// TIA Portal V19 program export: 1 tag tables, 1 data types, 3 data blocks, 8 code blocks (in call order from the OBs), 17 instance data blocks

VAR_GLOBAL   // PLC tag table "Default tag table"
   B0 AT %QB0 : Byte;
   B1 AT %QB1 : Byte;
   Clock_Byte AT %MB0 : Byte;
   Clock_10Hz AT %M0.0 : Bool;
   Clock_5Hz AT %M0.1 : Bool;
   "Clock_2.5Hz" AT %M0.2 : Bool;
   Clock_2Hz AT %M0.3 : Bool;
   "Clock_1.25Hz" AT %M0.4 : Bool;
   Clock_1Hz AT %M0.5 : Bool;
   "Clock_0.625Hz" AT %M0.6 : Bool;
   "Clock_0.5Hz" AT %M0.7 : Bool;
   System_Byte AT %MB1 : Byte;
   FirstScan AT %M1.0 : Bool;
   DiagStatusUpdate AT %M1.1 : Bool;
   AlwaysTRUE AT %M1.2 : Bool;
   AlwaysFALSE AT %M1.3 : Bool;
   "from et200sp PLC_1" AT %IB100 : Byte;
   toET200spfromPLC1 AT %QB100 : Byte;
   "from et200sp PLC_1 Right" AT %IB200 : Byte;
   "toET200spfromPLC1 Right" AT %QB200 : Byte;
END_VAR

TYPE "NetworkSwitchHMI"
   STRUCT
      Ports { S7_SetPoint := 'True'} : Array[1..8] of "LPNDR_typePortInformation";
      Port { S7_SetPoint := 'True'} : "LPNDR_typePortInformation";
      Index { S7_SetPoint := 'True'} : Int := 1;
   END_STRUCT;
END_TYPE

DATA_BLOCK "GlobalDB"   // DB9
{ S7_Optimized_Access := 'FALSE' }
   VAR RETAIN
      RTInfo : Struct   // Used to collect runtime information on an individual FB/FC
         Mode : UInt := 1;
         OBnumber : OB_ANY := 1;
         Info_LTIME : LTime := LT#0NS;
         RetVal : Int := 0;
      END_STRUCT;
      Runtime : Struct   // Used to collect individual runtime information of OB
         OB1Scan : Struct
            Min : LReal := 1000.0;
            Max : LReal;
            Current { ExternalAccessible := 'False'; ExternalVisible := 'False'; ExternalWritable := 'False'} : LReal;
            temp { ExternalAccessible := 'False'; ExternalVisible := 'False'; ExternalWritable := 'False'} : LReal;
            Mem { ExternalAccessible := 'False'; ExternalVisible := 'False'; ExternalWritable := 'False'} : LReal := 0.0;
            PreviousScan { ExternalAccessible := 'False'; ExternalVisible := 'False'; ExternalWritable := 'False'} : LReal;
            ResetMin : Bool;
            "Reset Max" : Bool;
         END_STRUCT;
      END_STRUCT;
      Trigger_StopSynch : Struct
         REQ_FullSwapSequence { S7_SetPoint := 'True'} : Bool;   // Trigger used to perform a full swap of PLCs
         REQ_StopPrimary { S7_SetPoint := 'True'} : Bool;   // trigger a primary stop
         REQ_SynchUp { S7_SetPoint := 'True'} : Bool;   // trigger a synchronization
         Mode_StopPrimary : Int := 8;   // Stop Primary = 8
         Mode_SynchUp : Int := 7;   // Synchronization = 7
         StopPrimary_Retry_Busy : Bool;   // triggered due to RHCTRL being busy
         SynchUp_Retry_Busy : Bool;   // triggered due to RHCTRL being busy
         SyncSequenceFlag : Bool;
         RH_CTRL_PrimaryStop : Struct   // Used to stop and synch primary or backup
            REQ : Bool;
            Ret_Val : Byte;
            Busy : Bool;
         END_STRUCT;
         RH_CTRL_SyncUp : Struct   // Used to stop and synch primary or backup
            REQ : Bool;
            Ret_Val : Byte;
            Busy : Bool;
         END_STRUCT;
         SyncSequenceTimer : IEC_TIMER;
         SequenceTimer : IEC_TIMER;   // Timer to sequence between stop and synch
         SequenceAlarm { S7_SetPoint := 'True'} : Bool;
      END_STRUCT;
      Network { S7_SetPoint := 'True'} : "NetworkSwitchHMI";
      SystemTime { S7_SetPoint := 'True'} : DTL;
      tempSystemTime { S7_SetPoint := 'True'} : Int;
   END_VAR
BEGIN
   Trigger_StopSynch.SequenceTimer.PT := T#25s;   // Time based on full sequence elapsed timer
END_DATA_BLOCK

DATA_BLOCK "hmiDatatransferTP1200"   // DB10
{ S7_Optimized_Access := 'TRUE' }
// stored: AutoNumber false, MemoryReserve 100
   VAR
      plc1LedState : Int;
      plc2LedState : Int;
      plcOperationState : Int;
      plcMrpState : Int;
      plcStopMonitoring : Int;
   END_VAR
BEGIN
END_DATA_BLOCK

DATA_BLOCK "DB_HMI Support"   // DB10000
{ S7_Optimized_Access := 'FALSE' }
// stored: AutoNumber false
   VAR
      "PLC Mode" : Int;
      "PLC Near Status" : Int;
      "PLC Far Status" : Int;
      "Bypasses Status" : Int;
      OperationStateSystem : Int;
      MRPRingState : Int;
   END_VAR
BEGIN
END_DATA_BLOCK

ORGANIZATION_BLOCK "Main"   // OB1, LAD, ProgramCycle
TITLE = "Main Program Sweep (Cycle)"
{ S7_Optimized_Access := 'TRUE' }
// stored: AutoNumber false, SetENOAutomatically false
   VAR_INPUT
      Initial_Call : Bool;   // Initial call of this OB
      Remanence : Bool;   // =True, if remanent data are available
   END_VAR
BEGIN

REGION Network 1: Map clock byte to output of dq card
   // Display "to" and "from" using move command for troubleshooting
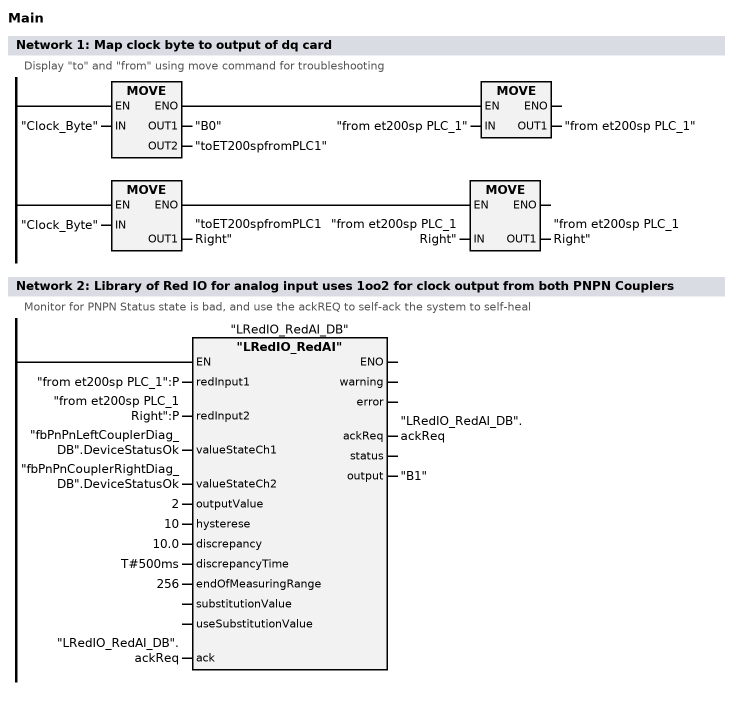
   RUNG wire#powerrail
      Move(in := "Clock_Byte", out1 => "B0", out2 => "toET200spfromPLC1")
      Move(in := "from et200sp PLC_1", out1 => "from et200sp PLC_1")
   END_RUNG
   RUNG wire#powerrail
      Move(in := "Clock_Byte", out1 => "toET200spfromPLC1 Right")
      Move(in := "from et200sp PLC_1 Right", out1 => "from et200sp PLC_1 Right")
   END_RUNG
   // the same network as SCL:
   "B0" := "Clock_Byte";
   "toET200spfromPLC1" := "Clock_Byte";
   "from et200sp PLC_1" := "from et200sp PLC_1";
   "toET200spfromPLC1 Right" := "Clock_Byte";
   "from et200sp PLC_1 Right" := "from et200sp PLC_1 Right";
END_REGION

REGION Network 2: Library of Red IO for analog input uses 1oo2 for clock output from both PNPN Couplers
   // Monitor for PNPN Status state is bad, and use the ackREQ to self-ack the system to self-heal
   RUNG wire#powerrail
      "LRedIO_RedAI_DB"(redInput1 := "from et200sp PLC_1":P, redInput2 := "from et200sp PLC_1 Right":P, valueStateCh1 := "fbPnPnLeftCouplerDiag_DB".DeviceStatusOk, valueStateCh2 := "fbPnPnCouplerRightDiag_DB".DeviceStatusOk, outputValue := 2, hysterese := 10, discrepancy := 10.0, discrepancyTime := T#500ms, endOfMeasuringRange := 256, substitutionValue :=, useSubstitutionValue :=, ack := "LRedIO_RedAI_DB".ackReq, warning =>, error =>, ackReq => "LRedIO_RedAI_DB".ackReq, status =>, output => "B1")
   END_RUNG
   // the same network as SCL:
   "LRedIO_RedAI_DB"(redInput1 := "from et200sp PLC_1":P,   // "LRedIO_RedAI"
                     redInput2 := "from et200sp PLC_1 Right":P,
                     valueStateCh1 := "fbPnPnLeftCouplerDiag_DB".DeviceStatusOk,
                     valueStateCh2 := "fbPnPnCouplerRightDiag_DB".DeviceStatusOk,
                     outputValue := 2,
                     hysterese := 10,
                     discrepancy := 10.0,
                     discrepancyTime := T#500ms,
                     endOfMeasuringRange := 256,
                     ack := "LRedIO_RedAI_DB".ackReq,
                     ackReq => "LRedIO_RedAI_DB".ackReq,
                     output => "B1");
END_REGION
END_ORGANIZATION_BLOCK

ORGANIZATION_BLOCK "Main_Switch"   // OB123, LAD, ProgramCycle
TITLE = "Main Program Sweep (Cycle)"
{ S7_Optimized_Access := 'TRUE' }
// stored: AutoNumber false, SetENOAutomatically false
   VAR_INPUT
      Initial_Call : Bool;   // Initial call of this OB
      Remanence : Bool;   // =True, if remanent data are available
   END_VAR
   VAR_TEMP
      retvalue : Int;
      text : String;
      retVal : Word;
      Busy : Bool;
   END_VAR
   VAR_TEMP   // added for the SCL form of the ladder/FBD networks
      _w1 : Bool;
   END_VAR
BEGIN

REGION Network 1: Cycle Measurement - Tic
   // Scan and store but only to reset the runtime counter at the top of the scan. the Ret_Val is collected at the end of the program cycle or area of focus.
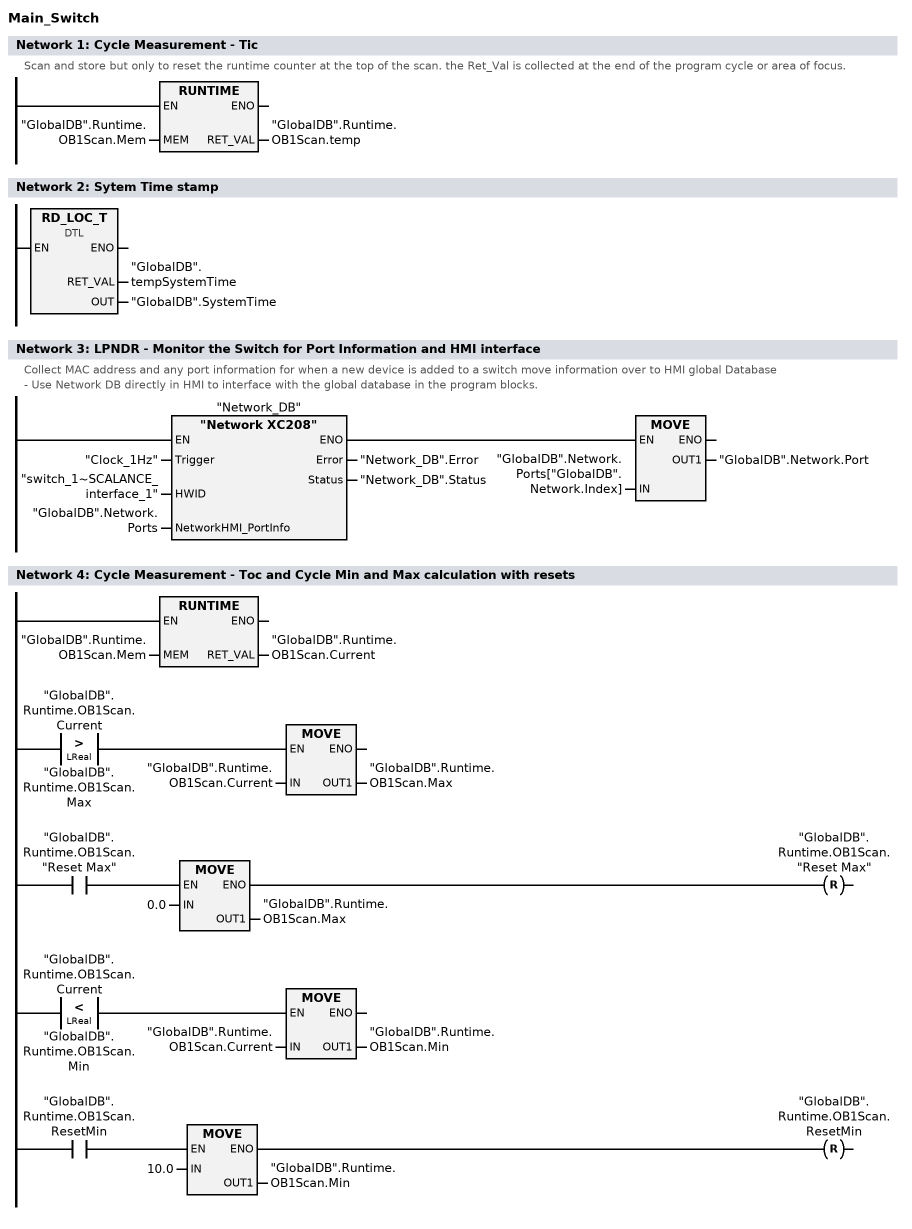
   // no SCL statement known for Runtime: written as a call
   "GlobalDB".Runtime.OB1Scan.temp := Runtime(mem := "GlobalDB".Runtime.OB1Scan.Mem);
END_REGION

REGION Network 2: Sytem Time stamp
   RUNG wire#powerrail
      { S7_Templates := "date_type := DTL" } RD_LOC_T(RET_VAL => "GlobalDB".tempSystemTime, OUT => "GlobalDB".SystemTime)
   END_RUNG
   // the same network as SCL:
   "GlobalDB".tempSystemTime := RD_LOC_T(OUT => "GlobalDB".SystemTime);
END_REGION

REGION Network 3: LPNDR - Monitor the Switch for Port Information and HMI interface
   // Collect MAC address and any port information for when a new device is added to a switch move information over to HMI global Database
   // 
   // - Use Network DB directly in HMI to interface with the global database in the program blocks.
   RUNG wire#powerrail
      "Network_DB"(Trigger := "Clock_1Hz", HWID := "switch_1~SCALANCE_interface_1", NetworkHMI_PortInfo := "GlobalDB".Network.Ports, Error => "Network_DB".Error, Status => "Network_DB".Status)
      Move(in := "GlobalDB".Network.Ports["GlobalDB".Network.Index], out1 => "GlobalDB".Network.Port)
   END_RUNG
   // the same network as SCL:
   "Network_DB"(Trigger := "Clock_1Hz",   // "Network XC208"
                HWID := "switch_1~SCALANCE_interface_1",
                NetworkHMI_PortInfo := "GlobalDB".Network.Ports,
                Error => "Network_DB".Error,
                Status => "Network_DB".Status,
                ENO => #_w1);
   IF #_w1 THEN "GlobalDB".Network.Port := "GlobalDB".Network.Ports["GlobalDB".Network.Index]; END_IF;
END_REGION

REGION Network 4: Cycle Measurement - Toc and Cycle Min and Max calculation with resets
   // no SCL statement known for Runtime: written as a call
   "GlobalDB".Runtime.OB1Scan.Current := Runtime(mem := "GlobalDB".Runtime.OB1Scan.Mem);
   IF "GlobalDB".Runtime.OB1Scan.Current > "GlobalDB".Runtime.OB1Scan.Max THEN
       "GlobalDB".Runtime.OB1Scan.Max := "GlobalDB".Runtime.OB1Scan.Current;
   END_IF;
   IF "GlobalDB".Runtime.OB1Scan."Reset Max" THEN
       "GlobalDB".Runtime.OB1Scan.Max := 0.0;
       "GlobalDB".Runtime.OB1Scan."Reset Max" := FALSE;
   END_IF;
   IF "GlobalDB".Runtime.OB1Scan.Current < "GlobalDB".Runtime.OB1Scan.Min THEN
       "GlobalDB".Runtime.OB1Scan.Min := "GlobalDB".Runtime.OB1Scan.Current;
   END_IF;
   IF "GlobalDB".Runtime.OB1Scan.ResetMin THEN
       "GlobalDB".Runtime.OB1Scan.Min := 10.0;
       "GlobalDB".Runtime.OB1Scan.ResetMin := FALSE;
   END_IF;
END_REGION
END_ORGANIZATION_BLOCK

FUNCTION_BLOCK "Network XC208"   // FB10, LAD
{ S7_Optimized_Access := 'TRUE' }
// stored: MemoryReserve 100, SetENOAutomatically false
   VAR_INPUT
      Trigger : Bool;   // Trigger the network scan for port info, rising edge
      HWID : HW_ANY;   // Scalance Interface of the switch
   END_VAR
   VAR_OUTPUT
      Error : Bool;
      Status : Word;
   END_VAR
   VAR_IN_OUT
      NetworkHMI_PortInfo : Variant;   // HMI input and output interface
   END_VAR
   VAR
      PortInformation { S7_SetPoint := 'True'} : "LPNDR_ReadGlobalInfo";   // LPNDR mode returns Port Information
   END_VAR
   VAR CONSTANT
      modeInterfaceInformation : Int := 1;
      modeMRPInformation : Int := 2;
      modePortInformation : Int := 3;
      modePortLinkStatus : Int := 4;
      modePortStatistics : Int := 5;
   END_VAR
BEGIN

REGION Network 1: Mode 3: Read Port Information
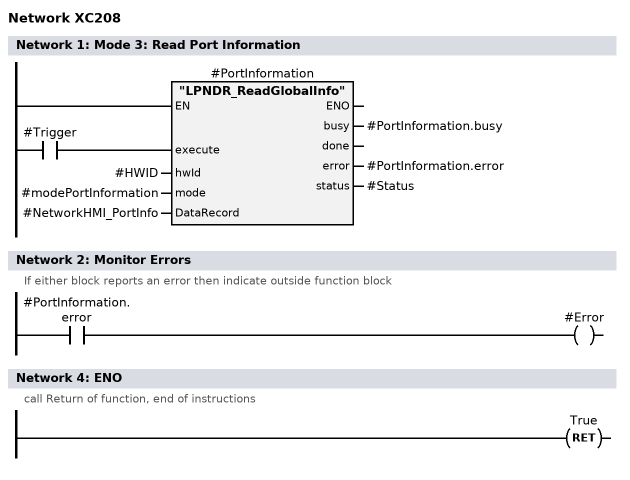
   RUNG wire#powerrail
      #PortInformation(execute := wire#w1, hwId := #HWID, mode := #modePortInformation, DataRecord := #NetworkHMI_PortInfo, busy => #PortInformation.busy, done =>, error => #PortInformation.error, status => #Status)
   END_RUNG
   RUNG wire#powerrail
      Contact( #Trigger )
   END_RUNG wire#w1
   // the same network as SCL:
   #PortInformation(execute := #Trigger,   // "LPNDR_ReadGlobalInfo"
                    hwId := #HWID,
                    mode := #modePortInformation,
                    DataRecord := #NetworkHMI_PortInfo,
                    busy => #PortInformation.busy,
                    error => #PortInformation.error,
                    status => #Status);
END_REGION

REGION Network 2: Monitor Errors
   // If either block reports an error then indicate outside function block
   RUNG wire#powerrail
      Contact( #PortInformation.error )
      Coil( #Error )
   END_RUNG
   // the same network as SCL:
   #Error := #PortInformation.error;
END_REGION

REGION Network 3
   // #Port."Port" := #Port.Ports[#Index];
END_REGION

REGION Network 4: ENO
   // call Return of function, end of instructions
   ENO := True;
   RETURN;
END_REGION
END_FUNCTION_BLOCK

ORGANIZATION_BLOCK "RT_Info_Cyclic"   // OB30, LAD, CyclicInterrupt
{ S7_Optimized_Access := 'TRUE' }
// stored: SetENOAutomatically false
   VAR_INPUT
      Initial_Call : Bool;   // Initial call of this OB
      Event_Count : Int;   // Events discarded
   END_VAR
   VAR CONSTANT
      constRunSoloState : Int := 37;
      constRunRedundant : Int := 40;
   END_VAR
   VAR_TEMP   // added for the SCL form of the ladder/FBD networks
      _w1 : Bool;
      _w2 : Bool;
      _w3 : Bool;
      _w4 : Bool;
   END_VAR
BEGIN

REGION Network 1: RT_Info for specific OB
   // Used to find the specific runtime of an OB, change the OB number and see the INFO.
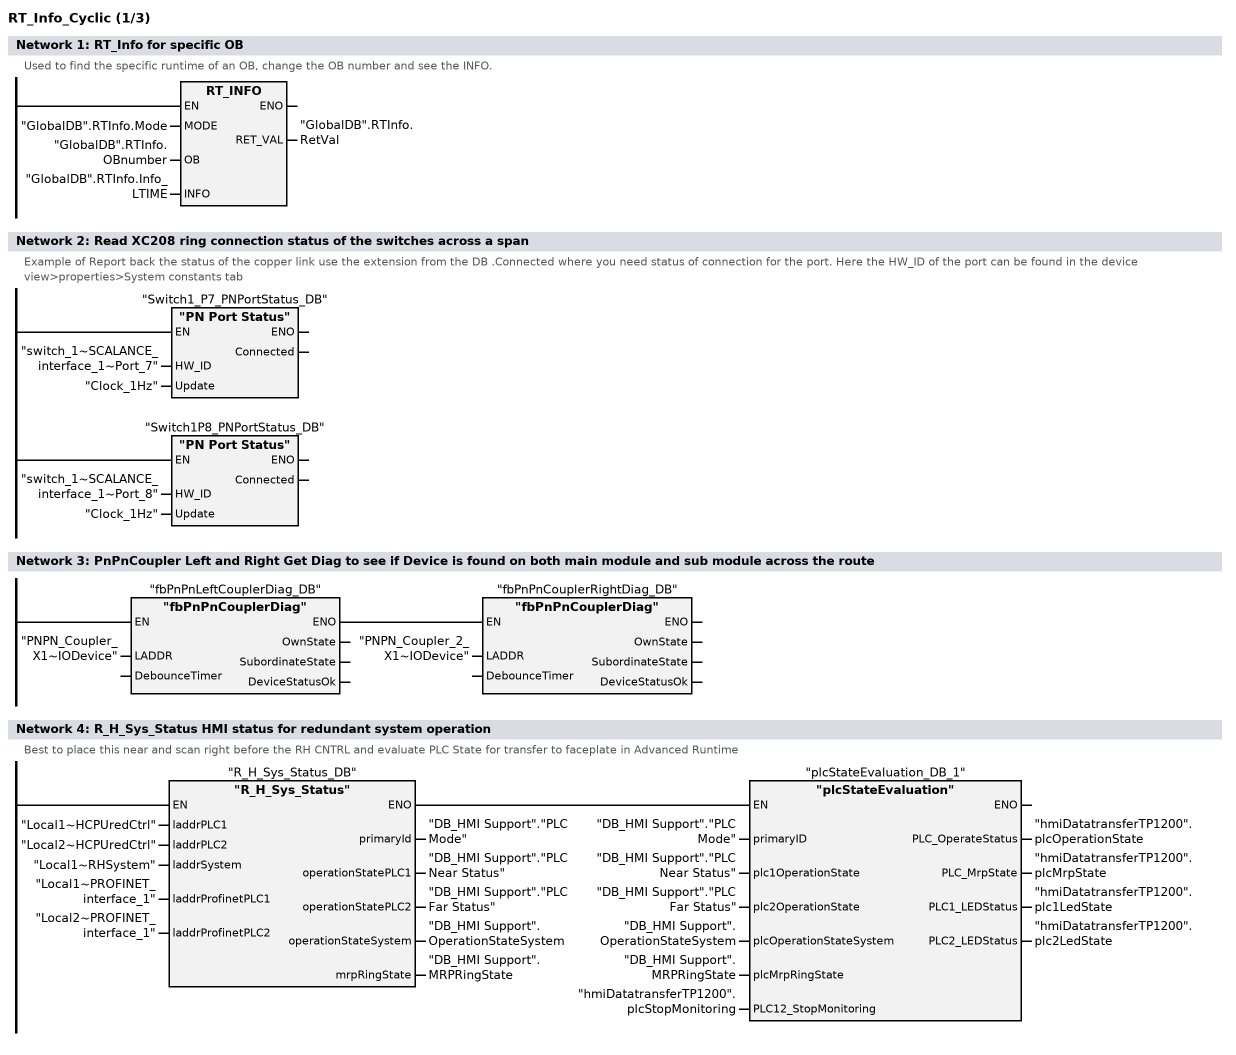
   RUNG wire#powerrail
      RT_INFO(MODE := "GlobalDB".RTInfo.Mode, OB := "GlobalDB".RTInfo.OBnumber, INFO := "GlobalDB".RTInfo.Info_LTIME, Ret_Val => "GlobalDB".RTInfo.RetVal)
   END_RUNG
   // the same network as SCL:
   "GlobalDB".RTInfo.RetVal := RT_INFO(MODE := "GlobalDB".RTInfo.Mode,
                           OB := "GlobalDB".RTInfo.OBnumber,
                           INFO := "GlobalDB".RTInfo.Info_LTIME);
END_REGION

REGION Network 2: Read XC208 ring connection status of the switches across a span
   // Example of Report back the status of the copper link use the extension from the DB .Connected where you need status of connection for the port. Here the HW_ID of the port can be found in the device view>properties>System constants tab
   RUNG wire#powerrail
      "Switch1_P7_PNPortStatus_DB"(HW_ID := "switch_1~SCALANCE_interface_1~Port_7", Update := "Clock_1Hz", Connected =>)
   END_RUNG
   RUNG wire#powerrail
      "Switch1P8_PNPortStatus_DB"(HW_ID := "switch_1~SCALANCE_interface_1~Port_8", Update := "Clock_1Hz", Connected =>)
   END_RUNG
   // the same network as SCL:
   "Switch1_P7_PNPortStatus_DB"(HW_ID := "switch_1~SCALANCE_interface_1~Port_7", Update := "Clock_1Hz");   // "PN Port Status"
   "Switch1P8_PNPortStatus_DB"(HW_ID := "switch_1~SCALANCE_interface_1~Port_8", Update := "Clock_1Hz");   // "PN Port Status"
END_REGION

REGION Network 3: PnPnCoupler Left and Right Get Diag to see if Device is found on both main module and sub module across the route
   RUNG wire#powerrail
      "fbPnPnLeftCouplerDiag_DB"(LADDR := "PNPN_Coupler_X1~IODevice", DebounceTimer :=, OwnState =>, SubordinateState =>, DeviceStatusOk =>)
      "fbPnPnCouplerRightDiag_DB"(LADDR := "PNPN_Coupler_2_X1~IODevice", DebounceTimer :=, OwnState =>, SubordinateState =>, DeviceStatusOk =>)
   END_RUNG
   // the same network as SCL:
   "fbPnPnLeftCouplerDiag_DB"(LADDR := "PNPN_Coupler_X1~IODevice", ENO => #_w1);   // "fbPnPnCouplerDiag"
   IF #_w1 THEN
       "fbPnPnCouplerRightDiag_DB"(LADDR := "PNPN_Coupler_2_X1~IODevice");   // "fbPnPnCouplerDiag"
   END_IF;
END_REGION

REGION Network 4: R_H_Sys_Status HMI status for redundant system operation
   // Best to place this near and scan right before the RH CNTRL and evaluate PLC State for transfer to faceplate in Advanced Runtime
   RUNG wire#powerrail
      "R_H_Sys_Status_DB"(laddrPLC1 := "Local1~HCPUredCtrl", laddrPLC2 := "Local2~HCPUredCtrl", laddrSystem := "Local1~RHSystem", laddrProfinetPLC1 := "Local1~PROFINET_interface_1", laddrProfinetPLC2 := "Local2~PROFINET_interface_1", primaryId => "DB_HMI Support"."PLC Mode", operationStatePLC1 => "DB_HMI Support"."PLC Near Status", operationStatePLC2 => "DB_HMI Support"."PLC Far Status", operationStateSystem => "DB_HMI Support".OperationStateSystem, mrpRingState => "DB_HMI Support".MRPRingState)
      "plcStateEvaluation_DB_1"(primaryID := "DB_HMI Support"."PLC Mode", plc1OperationState := "DB_HMI Support"."PLC Near Status", plc2OperationState := "DB_HMI Support"."PLC Far Status", plcOperationStateSystem := "DB_HMI Support".OperationStateSystem, plcMrpRingState := "DB_HMI Support".MRPRingState, PLC12_StopMonitoring := "hmiDatatransferTP1200".plcStopMonitoring, PLC_OperateStatus => "hmiDatatransferTP1200".plcOperationState, PLC_MrpState => "hmiDatatransferTP1200".plcMrpState, PLC1_LEDStatus => "hmiDatatransferTP1200".plc1LedState, PLC2_LEDStatus => "hmiDatatransferTP1200".plc2LedState)
   END_RUNG
   // the same network as SCL:
   "R_H_Sys_Status_DB"(laddrPLC1 := "Local1~HCPUredCtrl",   // "R_H_Sys_Status"
                       laddrPLC2 := "Local2~HCPUredCtrl",
                       laddrSystem := "Local1~RHSystem",
                       laddrProfinetPLC1 := "Local1~PROFINET_interface_1",
                       laddrProfinetPLC2 := "Local2~PROFINET_interface_1",
                       primaryId => "DB_HMI Support"."PLC Mode",
                       operationStatePLC1 => "DB_HMI Support"."PLC Near Status",
                       operationStatePLC2 => "DB_HMI Support"."PLC Far Status",
                       operationStateSystem => "DB_HMI Support".OperationStateSystem,
                       mrpRingState => "DB_HMI Support".MRPRingState,
                       ENO => #_w1);
   IF #_w1 THEN
       "plcStateEvaluation_DB_1"(primaryID := "DB_HMI Support"."PLC Mode",   // "plcStateEvaluation"
                               plc1OperationState := "DB_HMI Support"."PLC Near Status",
                               plc2OperationState := "DB_HMI Support"."PLC Far Status",
                               plcOperationStateSystem := "DB_HMI Support".OperationStateSystem,
                               plcMrpRingState := "DB_HMI Support".MRPRingState,
                               PLC12_StopMonitoring := "hmiDatatransferTP1200".plcStopMonitoring,
                               PLC_OperateStatus => "hmiDatatransferTP1200".plcOperationState,
                               PLC_MrpState => "hmiDatatransferTP1200".plcMrpState,
                               PLC1_LEDStatus => "hmiDatatransferTP1200".plc1LedState,
                               PLC2_LEDStatus => "hmiDatatransferTP1200".plc2LedState);
   END_IF;
END_REGION

REGION Network 5: Trigger primary stop RH_CNTRL
   // Self Latching Sequence using FullSwap Sequence tag, independent function with REQ tag
   // Used to trigger Primary Stop based on input from stop primary and full swap boolean tag;
   //  positive edge triggered instruction RH_CTRL below.
   // This network uses a Primary stop request, and evaluates if the RH_CTRL is busy before 
   // changing the mode or moving on to the next step.
   // The Retry_Busy tag is used to record if a Busy bit was in place while being triggered to prevent moving
   //  mode during middle of RH_CTRL operation.
   // 
   // Modes:
   // 3: Disable execution of the SYNCUP
   // 4: Re-enable execution of the SYNCUP
   // 7: Request SYNCUP system state 
   // 8: Request STOP of the primary CPU
   // 9: Request STOP of the backup CPU
   // 
   // Use mode 8 to stop the primary PLC, then use Mode 7 to Synch the primary and backup.
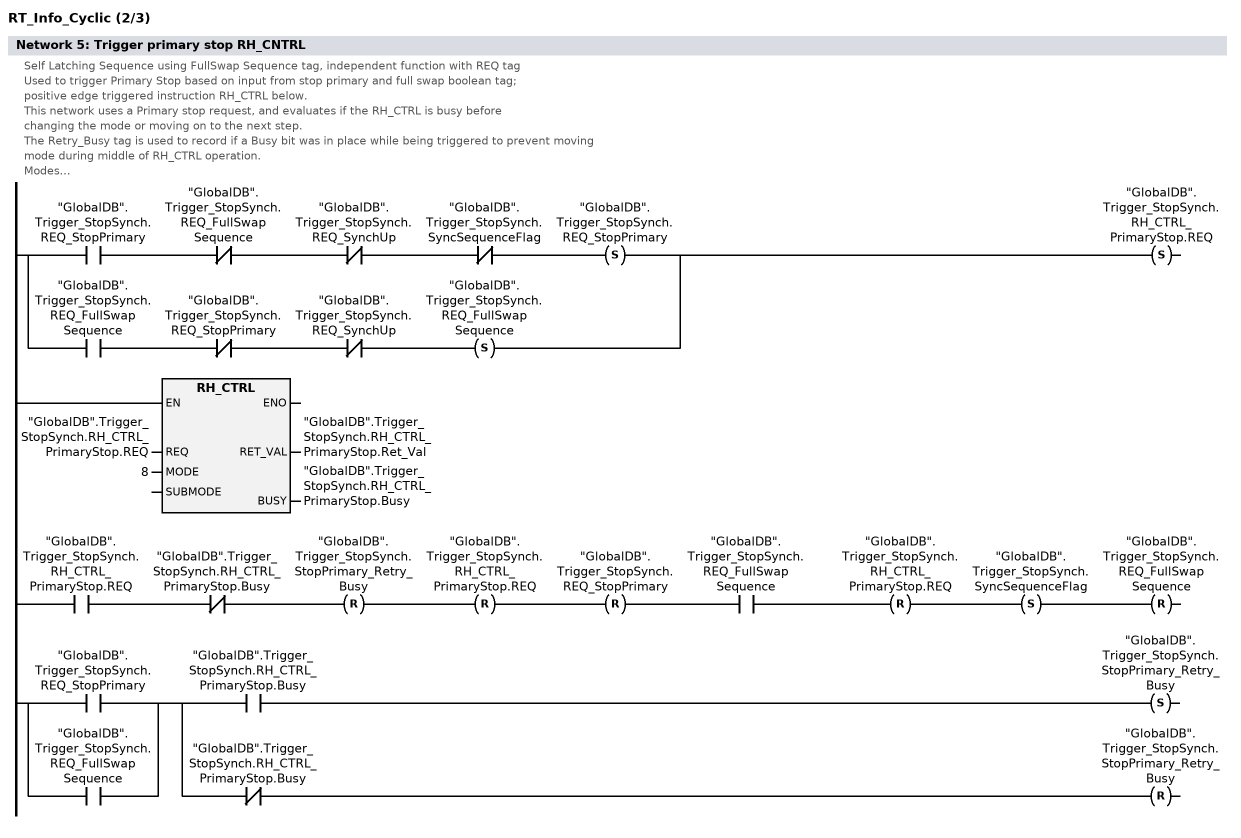
   RUNG wire#powerrail
      Contact( "GlobalDB".Trigger_StopSynch.REQ_StopPrimary )
      I_Contact( "GlobalDB".Trigger_StopSynch.REQ_FullSwapSequence )
      I_Contact( "GlobalDB".Trigger_StopSynch.REQ_SynchUp )
      I_Contact( "GlobalDB".Trigger_StopSynch.SyncSequenceFlag )
      S_Coil( "GlobalDB".Trigger_StopSynch.REQ_StopPrimary )
      wire#w1
      S_Coil( "GlobalDB".Trigger_StopSynch.RH_CTRL_PrimaryStop.REQ )
   END_RUNG
   RUNG wire#powerrail
      Contact( "GlobalDB".Trigger_StopSynch.REQ_FullSwapSequence )
      I_Contact( "GlobalDB".Trigger_StopSynch.REQ_StopPrimary )
      I_Contact( "GlobalDB".Trigger_StopSynch.REQ_SynchUp )
      S_Coil( "GlobalDB".Trigger_StopSynch.REQ_FullSwapSequence )
   END_RUNG wire#w1
   RUNG wire#powerrail
      RH_CTRL(REQ := "GlobalDB".Trigger_StopSynch.RH_CTRL_PrimaryStop.REQ, Mode := 8, Submode :=, Ret_Val => "GlobalDB".Trigger_StopSynch.RH_CTRL_PrimaryStop.Ret_Val, Busy => "GlobalDB".Trigger_StopSynch.RH_CTRL_PrimaryStop.Busy)
   END_RUNG
   RUNG wire#powerrail
      Contact( "GlobalDB".Trigger_StopSynch.RH_CTRL_PrimaryStop.REQ )
      I_Contact( "GlobalDB".Trigger_StopSynch.RH_CTRL_PrimaryStop.Busy )
      R_Coil( "GlobalDB".Trigger_StopSynch.StopPrimary_Retry_Busy )
      R_Coil( "GlobalDB".Trigger_StopSynch.RH_CTRL_PrimaryStop.REQ )
      R_Coil( "GlobalDB".Trigger_StopSynch.REQ_StopPrimary )
      Contact( "GlobalDB".Trigger_StopSynch.REQ_FullSwapSequence )
      R_Coil( "GlobalDB".Trigger_StopSynch.RH_CTRL_PrimaryStop.REQ )
      S_Coil( "GlobalDB".Trigger_StopSynch.SyncSequenceFlag )
      R_Coil( "GlobalDB".Trigger_StopSynch.REQ_FullSwapSequence )
   END_RUNG
   RUNG wire#powerrail
      Contact( "GlobalDB".Trigger_StopSynch.REQ_StopPrimary )
      wire#w2
      Contact( "GlobalDB".Trigger_StopSynch.RH_CTRL_PrimaryStop.Busy )
      S_Coil( "GlobalDB".Trigger_StopSynch.StopPrimary_Retry_Busy )
   END_RUNG
   RUNG wire#powerrail
      Contact( "GlobalDB".Trigger_StopSynch.REQ_FullSwapSequence )
   END_RUNG wire#w2
   RUNG wire#w2
      I_Contact( "GlobalDB".Trigger_StopSynch.RH_CTRL_PrimaryStop.Busy )
      R_Coil( "GlobalDB".Trigger_StopSynch.StopPrimary_Retry_Busy )
   END_RUNG
   // the same network as SCL:
   #_w1 := "GlobalDB".Trigger_StopSynch.REQ_StopPrimary AND NOT "GlobalDB".Trigger_StopSynch.REQ_FullSwapSequence AND NOT "GlobalDB".Trigger_StopSynch.REQ_SynchUp AND NOT "GlobalDB".Trigger_StopSynch.SyncSequenceFlag;
   IF #_w1 THEN "GlobalDB".Trigger_StopSynch.REQ_StopPrimary := TRUE; END_IF;
   #_w2 := "GlobalDB".Trigger_StopSynch.REQ_FullSwapSequence AND NOT "GlobalDB".Trigger_StopSynch.REQ_StopPrimary AND NOT "GlobalDB".Trigger_StopSynch.REQ_SynchUp;
   IF #_w2 THEN "GlobalDB".Trigger_StopSynch.REQ_FullSwapSequence := TRUE; END_IF;
   IF #_w1 OR #_w2 THEN "GlobalDB".Trigger_StopSynch.RH_CTRL_PrimaryStop.REQ := TRUE; END_IF;
   "GlobalDB".Trigger_StopSynch.RH_CTRL_PrimaryStop.Ret_Val := RH_CTRL(REQ := "GlobalDB".Trigger_StopSynch.RH_CTRL_PrimaryStop.REQ,
                           Mode := 8,
                           Busy => "GlobalDB".Trigger_StopSynch.RH_CTRL_PrimaryStop.Busy);
   #_w3 := "GlobalDB".Trigger_StopSynch.RH_CTRL_PrimaryStop.REQ AND NOT "GlobalDB".Trigger_StopSynch.RH_CTRL_PrimaryStop.Busy;
   IF #_w3 THEN
       "GlobalDB".Trigger_StopSynch.StopPrimary_Retry_Busy := FALSE;
       "GlobalDB".Trigger_StopSynch.RH_CTRL_PrimaryStop.REQ := FALSE;
       "GlobalDB".Trigger_StopSynch.REQ_StopPrimary := FALSE;
   END_IF;
   IF #_w3 AND "GlobalDB".Trigger_StopSynch.REQ_FullSwapSequence THEN
       "GlobalDB".Trigger_StopSynch.RH_CTRL_PrimaryStop.REQ := FALSE;
       "GlobalDB".Trigger_StopSynch.SyncSequenceFlag := TRUE;
       "GlobalDB".Trigger_StopSynch.REQ_FullSwapSequence := FALSE;
   END_IF;
   #_w4 := "GlobalDB".Trigger_StopSynch.REQ_StopPrimary OR "GlobalDB".Trigger_StopSynch.REQ_FullSwapSequence;
   IF #_w4 AND "GlobalDB".Trigger_StopSynch.RH_CTRL_PrimaryStop.Busy THEN
       "GlobalDB".Trigger_StopSynch.StopPrimary_Retry_Busy := TRUE;
   END_IF;
   IF #_w4 AND NOT "GlobalDB".Trigger_StopSynch.RH_CTRL_PrimaryStop.Busy THEN
       "GlobalDB".Trigger_StopSynch.StopPrimary_Retry_Busy := FALSE;
   END_IF;
END_REGION

REGION Network 6: Trigger Synch up RH_CNTRL
   // Self Latching Sequence using FullSwap Sequence tag, independent function with REQ tag
   // Used to trigger Sync up; positive edge triggered instruction RH_CTRL below
   // Sequence can also be triggered by Full sequence request which can set the SyncSequenceFlag below
   // SyncSequence Flag is help for next step until run Run-Solo status is reported
   //  positive edge triggered instruction RH_CTRL below
   // This network uses a synch up request, and evaluates if the RH_CTRL is busy before changing the mode
   // The Retry_Busy tag is used to record if a Busy bit was in place while being triggered to prevent moving
   //  mode during middle of RH_CTRL operation
   // 
   // Modes:
   // 3: Disable execution of the SYNCUP
   // 4: Re-enable execution of the SYNCUP
   // 7: Request SYNCUP system state 
   // 8: Request STOP of the primary CPU
   // 9: Request STOP of the backup CPU
   // 
   // Use mode 8 to stop the primary PLC, then use Mode 7 to Synch the primary and backup.
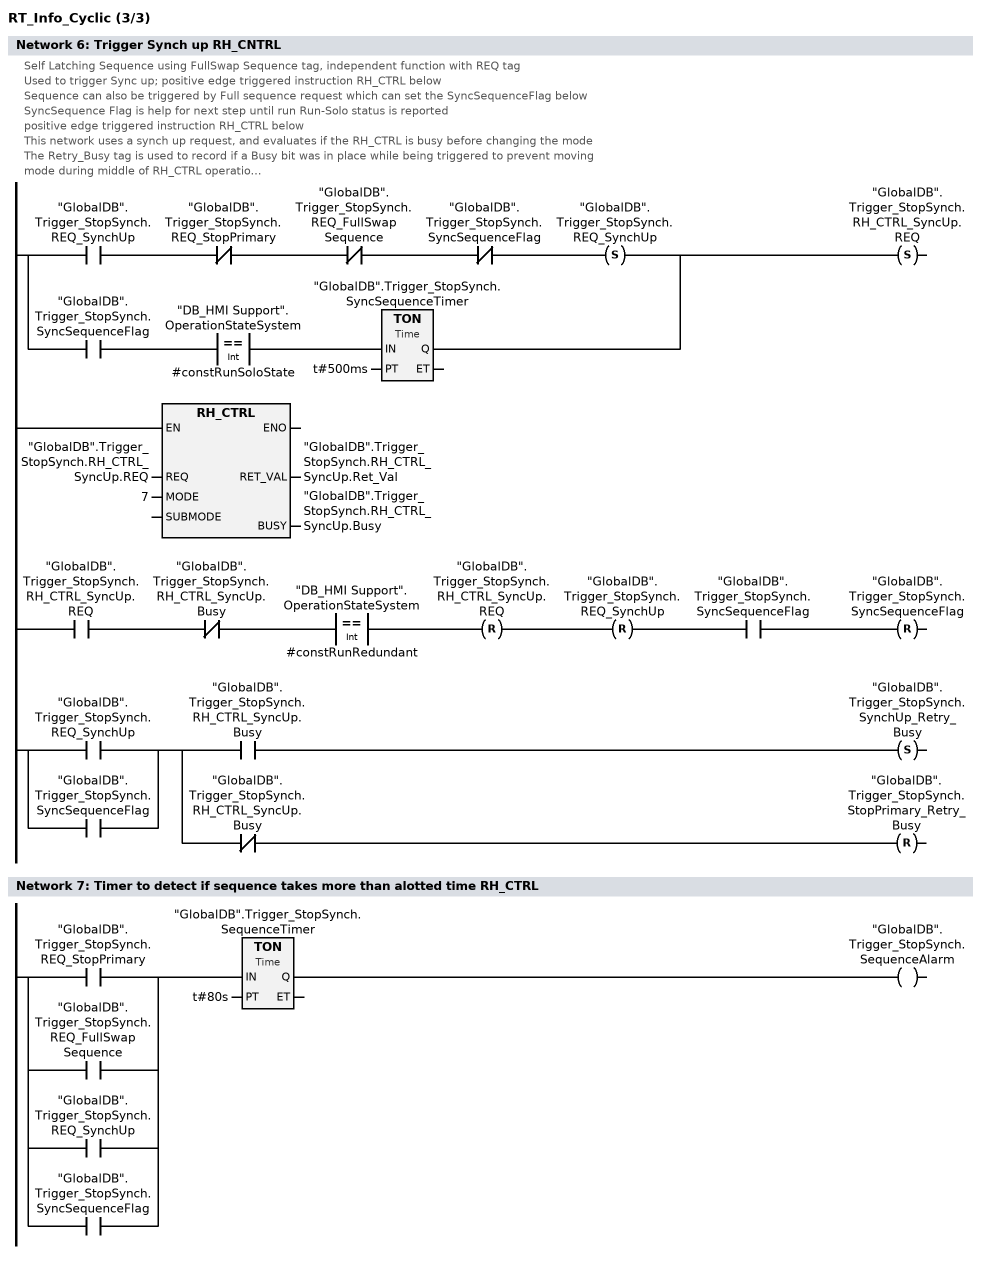
   RUNG wire#powerrail
      Contact( "GlobalDB".Trigger_StopSynch.REQ_SynchUp )
      I_Contact( "GlobalDB".Trigger_StopSynch.REQ_StopPrimary )
      I_Contact( "GlobalDB".Trigger_StopSynch.REQ_FullSwapSequence )
      I_Contact( "GlobalDB".Trigger_StopSynch.SyncSequenceFlag )
      S_Coil( "GlobalDB".Trigger_StopSynch.REQ_SynchUp )
      wire#w1
      S_Coil( "GlobalDB".Trigger_StopSynch.RH_CTRL_SyncUp.REQ )
   END_RUNG
   RUNG wire#powerrail
      Contact( "GlobalDB".Trigger_StopSynch.SyncSequenceFlag )
      { S7_Templates := "SrcType := Int" } EQ_Contact(in1 := "DB_HMI Support".OperationStateSystem, in2 := #constRunSoloState)
      { S7_Templates := "time_type := Time" } "GlobalDB".Trigger_StopSynch.SyncSequenceTimer.TON(pt := t#500ms, et =>)
   END_RUNG wire#w1
   RUNG wire#powerrail
      RH_CTRL(REQ := "GlobalDB".Trigger_StopSynch.RH_CTRL_SyncUp.REQ, Mode := 7, Submode :=, Ret_Val => "GlobalDB".Trigger_StopSynch.RH_CTRL_SyncUp.Ret_Val, Busy => "GlobalDB".Trigger_StopSynch.RH_CTRL_SyncUp.Busy)
   END_RUNG
   RUNG wire#powerrail
      Contact( "GlobalDB".Trigger_StopSynch.RH_CTRL_SyncUp.REQ )
      I_Contact( "GlobalDB".Trigger_StopSynch.RH_CTRL_SyncUp.Busy )
      { S7_Templates := "SrcType := Int" } EQ_Contact(in1 := "DB_HMI Support".OperationStateSystem, in2 := #constRunRedundant)
      R_Coil( "GlobalDB".Trigger_StopSynch.RH_CTRL_SyncUp.REQ )
      R_Coil( "GlobalDB".Trigger_StopSynch.REQ_SynchUp )
      Contact( "GlobalDB".Trigger_StopSynch.SyncSequenceFlag )
      R_Coil( "GlobalDB".Trigger_StopSynch.SyncSequenceFlag )
   END_RUNG
   RUNG wire#powerrail
      Contact( "GlobalDB".Trigger_StopSynch.REQ_SynchUp )
      wire#w2
      Contact( "GlobalDB".Trigger_StopSynch.RH_CTRL_SyncUp.Busy )
      S_Coil( "GlobalDB".Trigger_StopSynch.SynchUp_Retry_Busy )
   END_RUNG
   RUNG wire#powerrail
      Contact( "GlobalDB".Trigger_StopSynch.SyncSequenceFlag )
   END_RUNG wire#w2
   RUNG wire#w2
      I_Contact( "GlobalDB".Trigger_StopSynch.RH_CTRL_SyncUp.Busy )
      R_Coil( "GlobalDB".Trigger_StopSynch.StopPrimary_Retry_Busy )
   END_RUNG
   // the same network as SCL:
   #_w1 := "GlobalDB".Trigger_StopSynch.REQ_SynchUp AND NOT "GlobalDB".Trigger_StopSynch.REQ_StopPrimary AND NOT "GlobalDB".Trigger_StopSynch.REQ_FullSwapSequence AND NOT "GlobalDB".Trigger_StopSynch.SyncSequenceFlag;
   IF #_w1 THEN "GlobalDB".Trigger_StopSynch.REQ_SynchUp := TRUE; END_IF;
   "GlobalDB".Trigger_StopSynch.SyncSequenceTimer.TON(IN := "GlobalDB".Trigger_StopSynch.SyncSequenceFlag AND ("DB_HMI Support".OperationStateSystem = #constRunSoloState),
                           PT := t#500ms);
   IF #_w1 OR "GlobalDB".Trigger_StopSynch.SyncSequenceTimer.Q THEN
       "GlobalDB".Trigger_StopSynch.RH_CTRL_SyncUp.REQ := TRUE;
   END_IF;
   "GlobalDB".Trigger_StopSynch.RH_CTRL_SyncUp.Ret_Val := RH_CTRL(REQ := "GlobalDB".Trigger_StopSynch.RH_CTRL_SyncUp.REQ,
                           Mode := 7,
                           Busy => "GlobalDB".Trigger_StopSynch.RH_CTRL_SyncUp.Busy);
   #_w2 := "GlobalDB".Trigger_StopSynch.RH_CTRL_SyncUp.REQ AND NOT "GlobalDB".Trigger_StopSynch.RH_CTRL_SyncUp.Busy AND ("DB_HMI Support".OperationStateSystem = #constRunRedundant);
   IF #_w2 THEN
       "GlobalDB".Trigger_StopSynch.RH_CTRL_SyncUp.REQ := FALSE;
       "GlobalDB".Trigger_StopSynch.REQ_SynchUp := FALSE;
   END_IF;
   IF #_w2 AND "GlobalDB".Trigger_StopSynch.SyncSequenceFlag THEN
       "GlobalDB".Trigger_StopSynch.SyncSequenceFlag := FALSE;
   END_IF;
   #_w3 := "GlobalDB".Trigger_StopSynch.REQ_SynchUp OR "GlobalDB".Trigger_StopSynch.SyncSequenceFlag;
   IF #_w3 AND "GlobalDB".Trigger_StopSynch.RH_CTRL_SyncUp.Busy THEN
       "GlobalDB".Trigger_StopSynch.SynchUp_Retry_Busy := TRUE;
   END_IF;
   IF #_w3 AND NOT "GlobalDB".Trigger_StopSynch.RH_CTRL_SyncUp.Busy THEN
       "GlobalDB".Trigger_StopSynch.StopPrimary_Retry_Busy := FALSE;
   END_IF;
END_REGION

REGION Network 7: Timer to detect if sequence takes more than alotted time RH_CTRL
   RUNG wire#powerrail
      Contact( "GlobalDB".Trigger_StopSynch.REQ_StopPrimary )
      wire#w1
      { S7_Templates := "time_type := Time" } "GlobalDB".Trigger_StopSynch.SequenceTimer.TON(pt := t#80s, et =>)
      Coil( "GlobalDB".Trigger_StopSynch.SequenceAlarm )
   END_RUNG
   RUNG wire#powerrail
      Contact( "GlobalDB".Trigger_StopSynch.REQ_FullSwapSequence )
   END_RUNG wire#w1
   RUNG wire#powerrail
      Contact( "GlobalDB".Trigger_StopSynch.REQ_SynchUp )
   END_RUNG wire#w1
   RUNG wire#powerrail
      Contact( "GlobalDB".Trigger_StopSynch.SyncSequenceFlag )
   END_RUNG wire#w1
   // the same network as SCL:
   "GlobalDB".Trigger_StopSynch.SequenceTimer.TON(IN := "GlobalDB".Trigger_StopSynch.REQ_StopPrimary OR "GlobalDB".Trigger_StopSynch.REQ_FullSwapSequence OR "GlobalDB".Trigger_StopSynch.REQ_SynchUp OR "GlobalDB".Trigger_StopSynch.SyncSequenceFlag,
                           PT := t#80s);
   "GlobalDB".Trigger_StopSynch.SequenceAlarm := "GlobalDB".Trigger_StopSynch.SequenceTimer.Q;
END_REGION
END_ORGANIZATION_BLOCK

FUNCTION_BLOCK "PN Port Status"   // FB5, LAD
{ S7_Optimized_Access := 'TRUE' }
// stored: MemoryReserve 100, SetENOAutomatically false
   VAR_INPUT
      HW_ID : HW_IO;
      Update : Bool;
   END_VAR
   VAR_OUTPUT
      Connected : Bool;
   END_VAR
   VAR
      Updated_ReqP : Bool;
      Updated_Req : Bool;
      RDREC_Instance { S7_SetPoint := 'True'} : RDREC;
   END_VAR
   VAR_TEMP
      Record : Struct
         BlockType : Word;
         BlockLength : UInt;
         BlockVersionHigh : USInt;
         BlockVersionLow : USInt;
         Padding : Word;
         SlotNumber : Word;
         SubSlotNumber : Word;
         Data : Array[0..299] of Byte;
      END_STRUCT;
      n : Array[0..3] of UInt;
      LinkState : Word;
   END_VAR
   VAR_TEMP   // added for the SCL form of the ladder/FBD networks
      _w1 : Bool;
   END_VAR
BEGIN

REGION Network 1: Positive Edge triggered Update Req
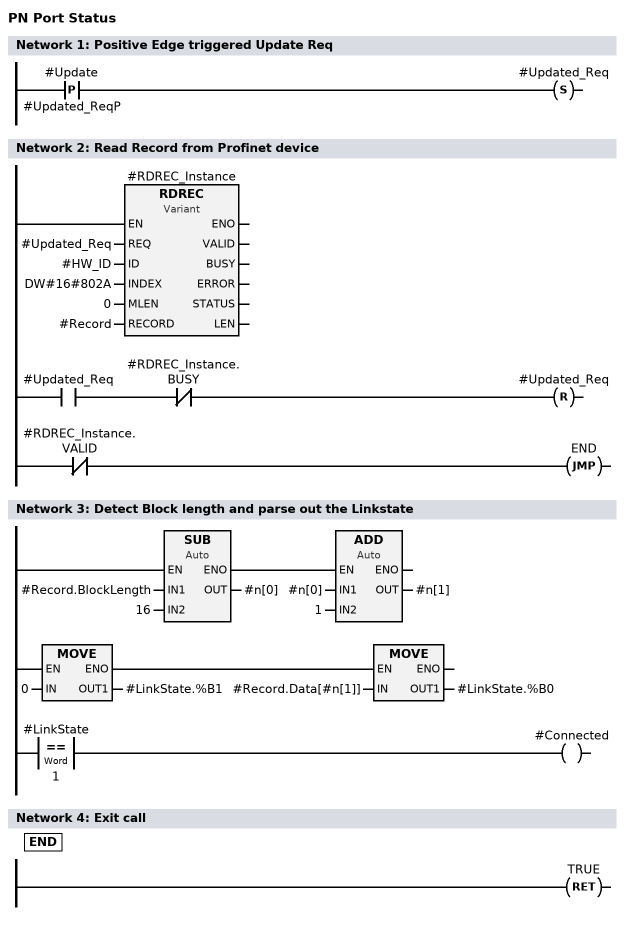
   RUNG wire#powerrail
      P_Contact(operand := #Update, bit := #Updated_ReqP)
      S_Coil( #Updated_Req )
   END_RUNG
   // the same network as SCL:
   #_w1 := #Update AND NOT #Updated_ReqP;   // rising edge of #Update
   #Updated_ReqP := #Update;
   IF #_w1 THEN #Updated_Req := TRUE; END_IF;
END_REGION

REGION Network 2: Read Record from Profinet device
   RUNG wire#powerrail
      { S7_Templates := "[ptr_type := Variant, id_type := HW_IO, index_type := DInt, len_type := UInt]" } #RDREC_Instance.RDREC(REQ := #Updated_Req, ID := #HW_ID, INDEX := DW#16#802A, MLEN := 0, RECORD := #Record, VALID =>, BUSY =>, ERROR =>, STATUS =>, LEN =>)
   END_RUNG
   RUNG wire#powerrail
      Contact( #Updated_Req )
      I_Contact( #RDREC_Instance.BUSY )
      R_Coil( #Updated_Req )
   END_RUNG
   RUNG wire#powerrail
      I_Contact( #RDREC_Instance.VALID )
      JumpCoil( END )
   END_RUNG
   // the same network as SCL:
   #RDREC_Instance(REQ := #Updated_Req, ID := #HW_ID, INDEX := DW#16#802A, MLEN := 0, RECORD := #Record);   // RDREC
   IF #Updated_Req AND NOT #RDREC_Instance.BUSY THEN #Updated_Req := FALSE; END_IF;
   IF NOT #RDREC_Instance.VALID THEN GOTO END; END_IF;
END_REGION

REGION Network 3: Detect Block length and parse out the Linkstate
   RUNG wire#powerrail
      Sub(in1 := #Record.BlockLength, in2 := 16, out => #n[0])
      Add(in1 := #n[0], in2 := 1, out => #n[1])
   END_RUNG
   RUNG wire#powerrail
      Move(in := 0, out1 => #LinkState.%B1)
      Move(in := #Record.Data[#n[1]], out1 => #LinkState.%B0)
   END_RUNG
   RUNG wire#powerrail
      { S7_Templates := "SrcType := Word" } EQ_Contact(in1 := #LinkState, in2 := 1)
      Coil( #Connected )
   END_RUNG
   // the same network as SCL:
   #n[0] := #Record.BlockLength - 16;
   #n[1] := #n[0] + 1;
   #LinkState.%B1 := 0;
   #LinkState.%B0 := #Record.Data[#n[1]];
   #Connected := #LinkState = 1;
END_REGION

REGION Network 4: Exit call
   END:
   ENO := TRUE;
   RETURN;
END_REGION
END_FUNCTION_BLOCK

FUNCTION_BLOCK "fbPnPnCouplerDiag"   // FB1, LAD
{ S7_Optimized_Access := 'TRUE' }
// stored: MemoryReserve 100, SetENOAutomatically false
   VAR_INPUT
      LADDR : HW_ANY;   // Hardware Address of the ~IODevice number
      DebounceTimer : Time := T#3ms;
   END_VAR
   VAR_OUTPUT
      OwnState : UInt;
      SubordinateState : UInt;
      DeviceStatusOk : Bool;
   END_VAR
   VAR
      Diag : DIS;
      Sub { S7_SetPoint := 'True'} : DNN;
      RetValueDiag : Int;
      CntDiagDiag : UInt;
      RetValueSub : Int;
      CntDiagSub : UInt;
      BadStateDebounceTimer : IEC_TIMER;
   END_VAR
   VAR CONSTANT
      "IO Device Mode" : Int := 1;
      "Subordinate device Mode" : Int := 2;
   END_VAR
   VAR_TEMP   // added for the SCL form of the ladder/FBD networks
      _w1 : Bool;
   END_VAR
BEGIN

REGION Network 1: PnPnCoupler Left Get Diag
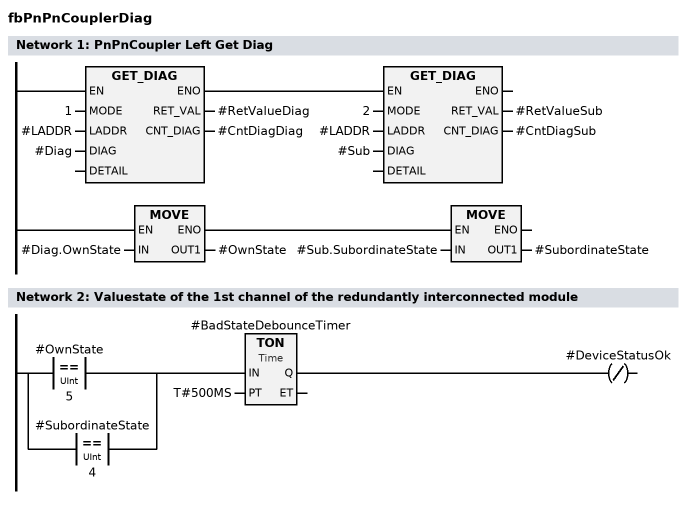
   RUNG wire#powerrail
      GET_DIAG(MODE := 1, LADDR := #LADDR, DIAG := #Diag, DETAIL :=, RET_VAL => #RetValueDiag, CNT_DIAG => #CntDiagDiag)
      GET_DIAG(MODE := 2, LADDR := #LADDR, DIAG := #Sub, DETAIL :=, RET_VAL => #RetValueSub, CNT_DIAG => #CntDiagSub)
   END_RUNG
   RUNG wire#powerrail
      Move(in := #Diag.OwnState, out1 => #OwnState)
      Move(in := #Sub.SubordinateState, out1 => #SubordinateState)
   END_RUNG
   // the same network as SCL:
   #RetValueDiag := GET_DIAG(MODE := 1, LADDR := #LADDR, DIAG := #Diag, CNT_DIAG => #CntDiagDiag, ENO => #_w1);
   IF #_w1 THEN
       #RetValueSub := GET_DIAG(MODE := 2, LADDR := #LADDR, DIAG := #Sub, CNT_DIAG => #CntDiagSub);
   END_IF;
   #OwnState := #Diag.OwnState;
   #SubordinateState := #Sub.SubordinateState;
END_REGION

REGION Network 2: Valuestate of the 1st channel of the redundantly interconnected module
   RUNG wire#powerrail
      { S7_Templates := "SrcType := UInt" } EQ_Contact(in1 := #OwnState, in2 := 5)
      wire#w1
      { S7_Templates := "time_type := Time" } #BadStateDebounceTimer.TON(pt := T#500MS, et =>)
      I_Coil( #DeviceStatusOk )
   END_RUNG
   RUNG wire#powerrail
      { S7_Templates := "SrcType := UInt" } EQ_Contact(in1 := #SubordinateState, in2 := 4)
   END_RUNG wire#w1
   // the same network as SCL:
   #BadStateDebounceTimer.TON(IN := (#OwnState = 5) OR (#SubordinateState = 4), PT := T#500MS);
   #DeviceStatusOk := NOT #BadStateDebounceTimer.Q;
END_REGION
END_FUNCTION_BLOCK

FUNCTION "Move MAC" : Void   // FC11, LAD
{ S7_Optimized_Access := 'TRUE' }
// stored: SetENOAutomatically false
   VAR_INPUT
      InMAC : Array[0..5] of Byte;
   END_VAR
   VAR_OUTPUT
      OutMAC : Array[0..5] of Byte;
   END_VAR
BEGIN

REGION Network 1
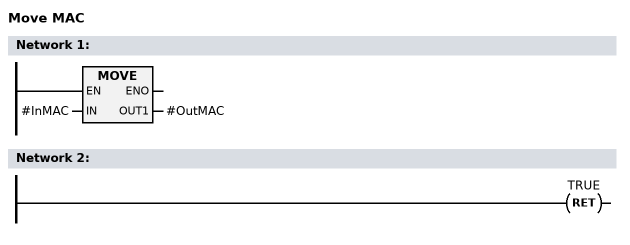
   RUNG wire#powerrail
      Move(in := #InMAC, out1 => #OutMAC)
   END_RUNG
   // the same network as SCL:
   #OutMAC := #InMAC;
END_REGION

REGION Network 2
   RUNG wire#powerrail
      ReturnCoil( TRUE )
   END_RUNG
   // the same network as SCL:
   ENO := TRUE;
   RETURN;
END_REGION
END_FUNCTION

FUNCTION_BLOCK "NetworkSwitchFaceplate"   // FB11, LAD
{ S7_Optimized_Access := 'TRUE' }
// stored: MemoryReserve 100, SetENOAutomatically false
   VAR_INPUT
      Index : Int;
   END_VAR
   VAR_OUTPUT
      PeerName { ExternalAccessible := 'False'; ExternalVisible := 'False'; ExternalWritable := 'False'} : String;
   END_VAR
   VAR_IN_OUT
      Port : "NetworkSwitchHMI";
   END_VAR
BEGIN

REGION Network 1 (SCL): Move all IN/OUT variables into Static values based on index selected from HMI

   #Port.Port := #Port.Ports[#Index];
END_REGION
END_FUNCTION_BLOCK

DATA_BLOCK "Network_DB"   // DB31
// stored: InstanceOfName Network XC208, InstanceOfType FB
"Network XC208"
BEGIN
END_DATA_BLOCK

DATA_BLOCK "PnPnLeftX2P1PNPortStatus_DB"   // DB11
// stored: InstanceOfName PN Port Status, InstanceOfType FB
"PN Port Status"
BEGIN
END_DATA_BLOCK

DATA_BLOCK "R_H_Sys_Status_DB"   // DB50
// stored: AutoNumber false, InstanceOfName R_H_Sys_Status, InstanceOfType FB
"R_H_Sys_Status"
   // VAR_INPUT
   //    laddrPLC1 : HW_ANY;
   //    laddrPLC2 : HW_ANY;
   //    laddrSystem : HW_ANY;
   //    laddrProfinetPLC1 : HW_ANY;
   //    laddrProfinetPLC2 : HW_ANY;
   // END_VAR
   // VAR_OUTPUT
   //    primaryId : Int;
   //    operationStatePLC1 : UInt;
   //    operationStatePLC2 : UInt;
   //    operationStateSystem : UInt;
   //    mrpRingState : UInt;
   // END_VAR
   // VAR
   //    statDiagModeCpu1 { S7_SetPoint := 'True'} : UInt;
   //    statCountDiagDetailsCpu1 : UInt;
   //    statReturnValueCpu1 : Int;
   //    statDiagCpu1 { ExternalAccessible := 'False'; ExternalVisible := 'False'; ExternalWritable := 'False'; S7_SetPoint := 'True'} : DIS;
   //    statDiagModeCpu2 { S7_SetPoint := 'True'} : UInt;
   //    statCountDiagDetailsCpu2 : UInt;
   //    statReturnValueCpu2 : Int;
   //    statDiagCpu2 { ExternalAccessible := 'False'; ExternalVisible := 'False'; ExternalWritable := 'False'; S7_SetPoint := 'True'} : DIS;
   //    statDiagModeSystem { S7_SetPoint := 'True'} : UInt;
   //    statCountDiagDetailsSystem : UInt;
   //    statReturnValueSystem : Int;
   //    statDiagSystem { ExternalAccessible := 'False'; ExternalVisible := 'False'; ExternalWritable := 'False'; S7_SetPoint := 'True'} : DIS;
   //    statDataRecord1 { S7_SetPoint := 'True'} : "LPNDR_typeMrpInformation";
   //    statDataRecord2 { S7_SetPoint := 'True'} : "LPNDR_typeMrpInformation";
   //    statLPNDR_ReadMrpState { S7_SetPoint := 'True'} : HW_ANY;
   //    statLPNDR_ReadGlobalInfo_DB1 { S7_SetPoint := 'True'} : "LPNDR_ReadGlobalInfo";
   //    statLPNDR_ReadGlobalInfo_DB2 { S7_SetPoint := 'True'} : "LPNDR_ReadGlobalInfo";
   //    statLPNDR_ReadMrpState_DB { S7_SetPoint := 'True'} : "LPNDR_ReadMrpState";
   //    statExecuteClock : Bool;
   //    IEC_Timer_0_Instance { S7_SetPoint := 'True'} : TOF_TIME;
   //    statToggleExecuteClock { S7_SetPoint := 'True'} : Bool;
   //    statUndefinedState : Bool;
   //    statExecuteClock2 : Bool;
   //    statToggleExecuteClock2 : Bool;
   //    IEC_Timer_0_Instance_1 { S7_SetPoint := 'True'} : TOF_TIME;
   //    IEC_Timer_0_Instance_2 { S7_SetPoint := 'True'} : TOF_TIME;
   //    statError1 : Bool;
   //    statChoose1 : Bool;
   //    IEC_Timer_0_Instance_3 { S7_SetPoint := 'True'} : TOF_TIME;
   //    statError2 : Bool;
   //    statChoose2 : Bool;
   // END_VAR
BEGIN
END_DATA_BLOCK

DATA_BLOCK "LPNDR_ReadGlobalInfo_Wlan1_DB"   // DB23
AUTHOR : SIOS
FAMILY : LPNDR
VERSION : 2.0
// stored: InstanceOfName LPNDR_ReadGlobalInfo_1, InstanceOfType FB
"LPNDR_ReadGlobalInfo_1"
   // VAR_INPUT
   //    execute : Bool;
   //    hwId : HW_IO;
   // END_VAR
   // VAR_OUTPUT
   //    done { ExternalWritable := 'False'} : Bool;
   //    busy { ExternalWritable := 'False'} : Bool;
   //    error { ExternalWritable := 'False'} : Bool;
   //    status { ExternalWritable := 'False'} : Word;
   //    InterfaceInformation : "LPNDR_typeInterfaceInformation";
   //    PortInformation : Array[1..52] of "LPNDR_typePortInformation";
   //    PortLinkState : Array[1..52] of "LPNDR_typePortLinkState";
   //    PortStatistic : Array[1..52] of "LPNDR_typePortStatistic";
   //    diagnostics { ExternalWritable := 'False'} : "typeDiagnostics";
   // END_VAR
   // VAR
   //    statExecuteOld { ExternalAccessible := 'False'; ExternalVisible := 'False'; ExternalWritable := 'False'} : Bool;
   //    statDone { ExternalAccessible := 'False'; ExternalVisible := 'False'; ExternalWritable := 'False'} : Bool;
   //    statBusy { ExternalAccessible := 'False'; ExternalVisible := 'False'; ExternalWritable := 'False'} : Bool;
   //    statError { ExternalAccessible := 'False'; ExternalVisible := 'False'; ExternalWritable := 'False'} : Bool;
   //    statStatus { ExternalAccessible := 'False'; ExternalVisible := 'False'; ExternalWritable := 'False'} : Word;
   //    statSubfunctionStatus { ExternalAccessible := 'False'; ExternalVisible := 'False'; ExternalWritable := 'False'} : Word;
   //    statFBErrorState { ExternalAccessible := 'False'; ExternalVisible := 'False'; ExternalWritable := 'False'} : DInt;
   //    statFBState { ExternalAccessible := 'False'; ExternalVisible := 'False'; ExternalWritable := 'False'} : DInt;
   //    statEmptyDiagnostics { ExternalAccessible := 'False'; ExternalVisible := 'False'; ExternalWritable := 'False'} : "typeDiagnostics";
   //    InstReadRecord { S7_SetPoint := 'True'} : RDREC;
   //    statReadRecordLength : UInt;
   //    statReadRecordRequest : Bool;
   //    statPDInterfaceMrpDataReal : UInt;
   //    statPDPortMrpDataReal : UInt;
   //    statPDInterfaceDataReal : UInt;
   //    statPDPortDataReal : UInt;
   //    statPDPortStatistic : UInt;
   //    statUnknown : UInt;
   //    statInterfaceInfoReset : "LPNDR_typeInterfaceInformation";
   //    statPortInfoReset { S7_SetPoint := 'True'} : "LPNDR_typePortInformation";
   //    statPortLinkStateReset { S7_SetPoint := 'True'} : "LPNDR_typePortLinkState";
   //    statPortStatisticReset { S7_SetPoint := 'True'} : "LPNDR_typePortStatistic";
   //    statReadRecord { S7_SetPoint := 'True'} : Array[0..4175] of Byte;
   // END_VAR
BEGIN
END_DATA_BLOCK

DATA_BLOCK "LPNDR_ReadGlobalInfo_Wlan2_DB"   // DB24
AUTHOR : SIOS
FAMILY : LPNDR
VERSION : 2.0
// stored: InstanceOfName LPNDR_ReadGlobalInfo_1, InstanceOfType FB
"LPNDR_ReadGlobalInfo_1"
   // VAR_INPUT
   //    execute : Bool;
   //    hwId : HW_IO;
   // END_VAR
   // VAR_OUTPUT
   //    done { ExternalWritable := 'False'} : Bool;
   //    busy { ExternalWritable := 'False'} : Bool;
   //    error { ExternalWritable := 'False'} : Bool;
   //    status { ExternalWritable := 'False'} : Word;
   //    InterfaceInformation : "LPNDR_typeInterfaceInformation";
   //    PortInformation : Array[1..52] of "LPNDR_typePortInformation";
   //    PortLinkState : Array[1..52] of "LPNDR_typePortLinkState";
   //    PortStatistic : Array[1..52] of "LPNDR_typePortStatistic";
   //    diagnostics { ExternalWritable := 'False'} : "typeDiagnostics";
   // END_VAR
   // VAR
   //    statExecuteOld { ExternalAccessible := 'False'; ExternalVisible := 'False'; ExternalWritable := 'False'} : Bool;
   //    statDone { ExternalAccessible := 'False'; ExternalVisible := 'False'; ExternalWritable := 'False'} : Bool;
   //    statBusy { ExternalAccessible := 'False'; ExternalVisible := 'False'; ExternalWritable := 'False'} : Bool;
   //    statError { ExternalAccessible := 'False'; ExternalVisible := 'False'; ExternalWritable := 'False'} : Bool;
   //    statStatus { ExternalAccessible := 'False'; ExternalVisible := 'False'; ExternalWritable := 'False'} : Word;
   //    statSubfunctionStatus { ExternalAccessible := 'False'; ExternalVisible := 'False'; ExternalWritable := 'False'} : Word;
   //    statFBErrorState { ExternalAccessible := 'False'; ExternalVisible := 'False'; ExternalWritable := 'False'} : DInt;
   //    statFBState { ExternalAccessible := 'False'; ExternalVisible := 'False'; ExternalWritable := 'False'} : DInt;
   //    statEmptyDiagnostics { ExternalAccessible := 'False'; ExternalVisible := 'False'; ExternalWritable := 'False'} : "typeDiagnostics";
   //    InstReadRecord { S7_SetPoint := 'True'} : RDREC;
   //    statReadRecordLength : UInt;
   //    statReadRecordRequest : Bool;
   //    statPDInterfaceMrpDataReal : UInt;
   //    statPDPortMrpDataReal : UInt;
   //    statPDInterfaceDataReal : UInt;
   //    statPDPortDataReal : UInt;
   //    statPDPortStatistic : UInt;
   //    statUnknown : UInt;
   //    statInterfaceInfoReset : "LPNDR_typeInterfaceInformation";
   //    statPortInfoReset { S7_SetPoint := 'True'} : "LPNDR_typePortInformation";
   //    statPortLinkStateReset { S7_SetPoint := 'True'} : "LPNDR_typePortLinkState";
   //    statPortStatisticReset { S7_SetPoint := 'True'} : "LPNDR_typePortStatistic";
   //    statReadRecord { S7_SetPoint := 'True'} : Array[0..4175] of Byte;
   // END_VAR
BEGIN
END_DATA_BLOCK

DATA_BLOCK "LPNDR_Readportinfo"   // DB33
// stored: InstanceOfName LPNDR_ReadGlobalInfo_2, InstanceOfType FB
"LPNDR_ReadGlobalInfo_2"
   // VAR_INPUT
   //    execute : Bool;
   //    hwId : HW_IO;
   //    mode : Int;
   // END_VAR
   // VAR_OUTPUT
   //    busy : Bool;
   //    done : Bool;
   //    error : Bool;
   //    status : Word;
   // END_VAR
   // VAR_IN_OUT
   //    DataRecord : Variant;
   // END_VAR
   // VAR
   //    InstReadRecord { S7_SetPoint := 'True'} : RDREC;
   //    statReadRecord { ExternalAccessible := 'False'; ExternalVisible := 'False'; ExternalWritable := 'False'} : Array[0..4175] of Byte;
   //    statReadRecordLength : UInt;
   //    statReadRecordRequest : Bool;
   //    statOldExecute : Bool;
   //    statPDInterfaceMrpDataReal : UInt;
   //    statPDPortMrpDataReal : UInt;
   //    statPDInterfaceDataReal : UInt;
   //    statPDPortDataReal : UInt;
   //    statPDPortStatistic : UInt;
   //    statUnknown : UInt;
   //    statInterfaceInformation { S7_SetPoint := 'True'} : "LPNDR_typeInterfaceInformation";
   //    statPortInformation { S7_SetPoint := 'True'} : Array[1..52] of "LPNDR_typePortInformation";
   //    statPortLinkState { S7_SetPoint := 'True'} : Array[1..52] of "LPNDR_typePortLinkState";
   //    statPortStatistic { S7_SetPoint := 'True'} : Array[1..52] of "LPNDR_typePortStatistic";
   //    statBusy { S7_SetPoint := 'True'} : Bool;
   // END_VAR
BEGIN
END_DATA_BLOCK

DATA_BLOCK "NetworkSwitchFaceplate_DB"   // DB32
// stored: InstanceOfName NetworkSwitchFaceplate, InstanceOfType FB
"NetworkSwitchFaceplate"
BEGIN
END_DATA_BLOCK

DATA_BLOCK "fbPnPnCouplerRightDiag_DB"   // DB12
// stored: InstanceOfName fbPnPnCouplerDiag, InstanceOfType FB
"fbPnPnCouplerDiag"
BEGIN
END_DATA_BLOCK

DATA_BLOCK "fbPnPnLeftCouplerDiag_DB"   // DB13
// stored: InstanceOfName fbPnPnCouplerDiag, InstanceOfType FB
"fbPnPnCouplerDiag"
BEGIN
END_DATA_BLOCK

DATA_BLOCK "instanceR_H_Sys_Status_DB"   // DB28
// stored: InstanceOfName R_H_Sys_Status, InstanceOfType FB
"R_H_Sys_Status"
   // VAR_INPUT
   //    laddrPLC1 : HW_ANY;
   //    laddrPLC2 : HW_ANY;
   //    laddrSystem : HW_ANY;
   //    laddrProfinetPLC1 : HW_ANY;
   //    laddrProfinetPLC2 : HW_ANY;
   // END_VAR
   // VAR_OUTPUT
   //    primaryId : Int;
   //    operationStatePLC1 : UInt;
   //    operationStatePLC2 : UInt;
   //    operationStateSystem : UInt;
   //    mrpRingState : UInt;
   // END_VAR
   // VAR
   //    statDiagModeCpu1 { S7_SetPoint := 'True'} : UInt;
   //    statCountDiagDetailsCpu1 : UInt;
   //    statReturnValueCpu1 : Int;
   //    statDiagCpu1 { ExternalAccessible := 'False'; ExternalVisible := 'False'; ExternalWritable := 'False'; S7_SetPoint := 'True'} : DIS;
   //    statDiagModeCpu2 { S7_SetPoint := 'True'} : UInt;
   //    statCountDiagDetailsCpu2 : UInt;
   //    statReturnValueCpu2 : Int;
   //    statDiagCpu2 { ExternalAccessible := 'False'; ExternalVisible := 'False'; ExternalWritable := 'False'; S7_SetPoint := 'True'} : DIS;
   //    statDiagModeSystem { S7_SetPoint := 'True'} : UInt;
   //    statCountDiagDetailsSystem : UInt;
   //    statReturnValueSystem : Int;
   //    statDiagSystem { ExternalAccessible := 'False'; ExternalVisible := 'False'; ExternalWritable := 'False'; S7_SetPoint := 'True'} : DIS;
   //    statDataRecord1 { S7_SetPoint := 'True'} : "LPNDR_typeMrpInformation";
   //    statDataRecord2 { S7_SetPoint := 'True'} : "LPNDR_typeMrpInformation";
   //    statLPNDR_ReadMrpState { S7_SetPoint := 'True'} : HW_ANY;
   //    statLPNDR_ReadGlobalInfo_DB1 { S7_SetPoint := 'True'} : "LPNDR_ReadGlobalInfo";
   //    statLPNDR_ReadGlobalInfo_DB2 { S7_SetPoint := 'True'} : "LPNDR_ReadGlobalInfo";
   //    statLPNDR_ReadMrpState_DB { S7_SetPoint := 'True'} : "LPNDR_ReadMrpState";
   //    statExecuteClock : Bool;
   //    IEC_Timer_0_Instance { S7_SetPoint := 'True'} : TOF_TIME;
   //    statToggleExecuteClock { S7_SetPoint := 'True'} : Bool;
   //    statUndefinedState : Bool;
   //    statExecuteClock2 : Bool;
   //    statToggleExecuteClock2 : Bool;
   //    IEC_Timer_0_Instance_1 { S7_SetPoint := 'True'} : TOF_TIME;
   //    IEC_Timer_0_Instance_2 { S7_SetPoint := 'True'} : TOF_TIME;
   //    statError1 : Bool;
   //    statChoose1 : Bool;
   //    IEC_Timer_0_Instance_3 { S7_SetPoint := 'True'} : TOF_TIME;
   //    statError2 : Bool;
   //    statChoose2 : Bool;
   // END_VAR
BEGIN
END_DATA_BLOCK

DATA_BLOCK "plcStateEvaluation_DB"   // DB27
// stored: InstanceOfName plcStateEvaluation, InstanceOfType FB
"plcStateEvaluation"
   // VAR_INPUT
   //    primaryID : Int;
   //    plc1OperationState : UInt;
   //    plc2OperationState : UInt;
   //    plcOperationStateSystem : UInt;
   //    plcMrpRingState : UInt;
   // END_VAR
   // VAR_OUTPUT
   //    PLC_OperateStatus : Int;
   //    PLC_MrpState : Int;
   //    PLC1_LEDStatus : Int;
   //    PLC2_LEDStatus : Int;
   // END_VAR
   // VAR_IN_OUT
   //    PLC12_StopMonitoring : Int;
   // END_VAR
   // VAR
   //    statPrimaryID : Int;
   //    statPlc1State : UInt;
   //    statPlc2State : UInt;
   //    statPlcStateSystem : UInt;
   //    statPlcMrpRingState : UInt;
   //    statPlcStatus : Int;
   //    statPLC12StopMonitoring : Int;
   // END_VAR
BEGIN
END_DATA_BLOCK

DATA_BLOCK "plcStateEvaluation_DB_1"   // DB29
// stored: InstanceOfName plcStateEvaluation, InstanceOfType FB
"plcStateEvaluation"
   // VAR_INPUT
   //    primaryID : Int;
   //    plc1OperationState : UInt;
   //    plc2OperationState : UInt;
   //    plcOperationStateSystem : UInt;
   //    plcMrpRingState : UInt;
   // END_VAR
   // VAR_OUTPUT
   //    PLC_OperateStatus : Int;
   //    PLC_MrpState : Int;
   //    PLC1_LEDStatus : Int;
   //    PLC2_LEDStatus : Int;
   // END_VAR
   // VAR_IN_OUT
   //    PLC12_StopMonitoring : Int;
   // END_VAR
   // VAR
   //    statPrimaryID : Int;
   //    statPlc1State : UInt;
   //    statPlc2State : UInt;
   //    statPlcStateSystem : UInt;
   //    statPlcMrpRingState : UInt;
   //    statPlcStatus : Int;
   //    statPLC12StopMonitoring : Int;
   // END_VAR
BEGIN
END_DATA_BLOCK

DATA_BLOCK "FBR1_PNPortStatus_DB"   // DB25
// stored: InstanceOfName PN Port Status, InstanceOfType FB
"PN Port Status"
BEGIN
END_DATA_BLOCK

DATA_BLOCK "FBR2_PNPortStatus_DB"   // DB26
// stored: InstanceOfName PN Port Status, InstanceOfType FB
"PN Port Status"
BEGIN
END_DATA_BLOCK

DATA_BLOCK "Switch1P8_PNPortStatus_DB"   // DB20
// stored: InstanceOfName PN Port Status, InstanceOfType FB
"PN Port Status"
BEGIN
END_DATA_BLOCK

DATA_BLOCK "Switch1_P7_PNPortStatus_DB"   // DB30
// stored: InstanceOfName PN Port Status, InstanceOfType FB
"PN Port Status"
BEGIN
END_DATA_BLOCK

DATA_BLOCK "LRedIO_RedAI_DB"   // DB1
AUTHOR : SiemensAG
FAMILY : LRedIO
VERSION : 1.0
// stored: InstanceOfName LRedIO_RedAI, InstanceOfType FB
"LRedIO_RedAI"
   // VAR_INPUT
   //    redInput1 : DInt;
   //    redInput2 : DInt;
   //    valueStateCh1 : Bool;
   //    valueStateCh2 : Bool;
   //    outputValue : USInt;
   //    hysterese : Int;
   //    discrepancy : Real;
   //    discrepancyTime : Time;
   //    endOfMeasuringRange : DInt;
   //    substitutionValue : DInt;
   //    useSubstitutionValue : USInt;
   //    ack : Bool;
   // END_VAR
   // VAR_OUTPUT
   //    warning : Bool;
   //    error : Bool;
   //    ackReq : Bool;
   //    status : Word;
   //    output : DInt;
   // END_VAR
   // VAR
   //    statRedInput1 { ExternalAccessible := 'False'; ExternalVisible := 'False'; ExternalWritable := 'False'} : DInt;
   //    statRedInput2 { ExternalAccessible := 'False'; ExternalVisible := 'False'; ExternalWritable := 'False'} : DInt;
   //    statValuestateCh1 { ExternalAccessible := 'False'; ExternalVisible := 'False'; ExternalWritable := 'False'} : Bool;
   //    statValuestateCh2 { ExternalAccessible := 'False'; ExternalVisible := 'False'; ExternalWritable := 'False'} : Bool;
   //    statDiscrepancy { ExternalAccessible := 'False'; ExternalVisible := 'False'; ExternalWritable := 'False'} : Real;
   //    statValuestateBad1 { ExternalAccessible := 'False'; ExternalVisible := 'False'; ExternalWritable := 'False'} : Bool;
   //    statValuestateBad2 { ExternalAccessible := 'False'; ExternalVisible := 'False'; ExternalWritable := 'False'} : Bool;
   //    statAck { ExternalAccessible := 'False'; ExternalVisible := 'False'; ExternalWritable := 'False'} : Bool;
   //    statAckNec { ExternalAccessible := 'False'; ExternalVisible := 'False'; ExternalWritable := 'False'} : Bool;
   //    statState { ExternalAccessible := 'False'; ExternalVisible := 'False'; ExternalWritable := 'False'} : Int;
   //    statDiscError { ExternalAccessible := 'False'; ExternalVisible := 'False'; ExternalWritable := 'False'} : Bool;
   //    statOutputValue { ExternalAccessible := 'False'; ExternalVisible := 'False'; ExternalWritable := 'False'} : USInt;
   //    statWrongOutputValue { ExternalAccessible := 'False'; ExternalVisible := 'False'; ExternalWritable := 'False'} : Bool;
   //    statWrongDisc { ExternalAccessible := 'False'; ExternalVisible := 'False'; ExternalWritable := 'False'} : Bool;
   //    statWrongHysterese { ExternalAccessible := 'False'; ExternalVisible := 'False'; ExternalWritable := 'False'} : Bool;
   //    statHysterese { ExternalAccessible := 'False'; ExternalVisible := 'False'; ExternalWritable := 'False'} : Int;
   //    statInputDifference { ExternalAccessible := 'False'; ExternalVisible := 'False'; ExternalWritable := 'False'} : DInt;
   //    statAbsInputDifference { ExternalAccessible := 'False'; ExternalVisible := 'False'; ExternalWritable := 'False'} : DInt;
   //    statDiscrepancyCalc { ExternalAccessible := 'False'; ExternalVisible := 'False'; ExternalWritable := 'False'} : DInt;
   //    statHystereseCalc { ExternalAccessible := 'False'; ExternalVisible := 'False'; ExternalWritable := 'False'} : DInt;
   //    statHysteresecheckOK { ExternalAccessible := 'False'; ExternalVisible := 'False'; ExternalWritable := 'False'} : Bool;
   //    statEndOfMeasuringRange { ExternalAccessible := 'False'; ExternalVisible := 'False'; ExternalWritable := 'False'} : DInt;
   //    statWrongEndOfMeasuringRange { ExternalAccessible := 'False'; ExternalVisible := 'False'; ExternalWritable := 'False'} : Bool;
   //    statSubValue { ExternalAccessible := 'False'; ExternalVisible := 'False'; ExternalWritable := 'False'} : DInt;
   //    statUseSubstitutionValue { ExternalAccessible := 'False'; ExternalVisible := 'False'; ExternalWritable := 'False'} : USInt;
   //    statWrongSubValue { ExternalAccessible := 'False'; ExternalVisible := 'False'; ExternalWritable := 'False'} : Bool;
   //    statAckEdge { ExternalAccessible := 'False'; ExternalVisible := 'False'; ExternalWritable := 'False'} : Bool;
   //    statWrongUseSubVal { ExternalAccessible := 'False'; ExternalVisible := 'False'; ExternalWritable := 'False'} : Bool;
   //    statDiscrepancyTime { ExternalAccessible := 'False'; ExternalVisible := 'False'; ExternalWritable := 'False'} : Time;
   //    statStartDiscTime { ExternalAccessible := 'False'; ExternalVisible := 'False'; ExternalWritable := 'False'} : Bool;
   //    statInstDiscrepancyTime { ExternalAccessible := 'False'; ExternalVisible := 'False'; ExternalWritable := 'False'; S7_SetPoint := 'True'} : TON_TIME;
   //    statStatus { ExternalAccessible := 'False'; ExternalVisible := 'False'; ExternalWritable := 'False'} : Word;
   //    statWrongDiscTime { ExternalAccessible := 'False'; ExternalVisible := 'False'; ExternalWritable := 'False'} : Bool;
   //    statOutput { ExternalAccessible := 'False'; ExternalVisible := 'False'; ExternalWritable := 'False'} : DInt;
   //    statParamError { ExternalAccessible := 'False'; ExternalVisible := 'False'; ExternalWritable := 'False'} : Bool;
   //    statOldRedInput1 { ExternalAccessible := 'False'; ExternalVisible := 'False'; ExternalWritable := 'False'} : DInt;
   //    statOldRedInput2 { ExternalAccessible := 'False'; ExternalVisible := 'False'; ExternalWritable := 'False'} : DInt;
   //    statNewRedInput1 { ExternalAccessible := 'False'; ExternalVisible := 'False'; ExternalWritable := 'False'} : DInt;
   //    statNewRedInput2 { ExternalAccessible := 'False'; ExternalVisible := 'False'; ExternalWritable := 'False'} : DInt;
   //    statLastValidOut { ExternalAccessible := 'False'; ExternalVisible := 'False'; ExternalWritable := 'False'} : DInt;
   //    statStoreRisingEdge : Bool;
   //    statDiscrepancyTimeTrue : Bool;
   // END_VAR
BEGIN
END_DATA_BLOCK
